{attribute 'linkalways'} 
{attribute 'no_explicit_call' := 'This FB is a CLASS and must be accessed using methods or properties'}
{attribute 'enable_dynamic_creation'}
FUNCTION_BLOCK FINAL GT_DWORD EXTENDS Node
VAR
	in1 : _DWORD(0);
	in2 : _DWORD(0);
	out : _BOOL(FALSE);
END_VAR

METHOD PUBLIC Clone : I_Node
VAR
	pNode : POINTER TO GT_DWORD;
END_VAR
pNode := __NEW(GT_DWORD);
Clone := pNode^;
END_METHOD

METHOD FB_init : BOOL
VAR_INPUT
	bInitRetains : BOOL; // if TRUE, the retain variables are initialized (warm start / cold start)
	bInCopyCode : BOOL;  // if TRUE, the instance afterwards gets moved into the copy code (online change)
END_VAR
AddInput('in1',THIS^.in1);
AddInput('in2',THIS^.in2);
AddOutput('out', THIS^.out);
END_METHOD

METHOD PROTECTED OnExecute
VAR
END_VAR
out.Value := in1.Value > in2.Value;
END_METHOD

END_FUNCTION_BLOCK

(* stored: Version 1.1.0.1, ProductVersion 3.1.4024.15
   POU GT_DWORD: Id {6cd531d7-1cfa-4c54-aab0-1a6927c96654}, SpecialFunc None
   Folder Constructor: Id {db5c64d8-7ee4-49ab-8eae-61afc1989cca}
   Method Clone: Id {a30e38ed-5244-4ea5-ba3e-ac0f93098b03}
   Method FB_init: Id {eda2d975-a3af-4889-8914-a21dcfef8892}
   Method OnExecute: Id {18b6cd86-b8f6-4464-8529-a358b44070a2} *)
